RoboDK station: kr30 cnc 042619 3.rdk

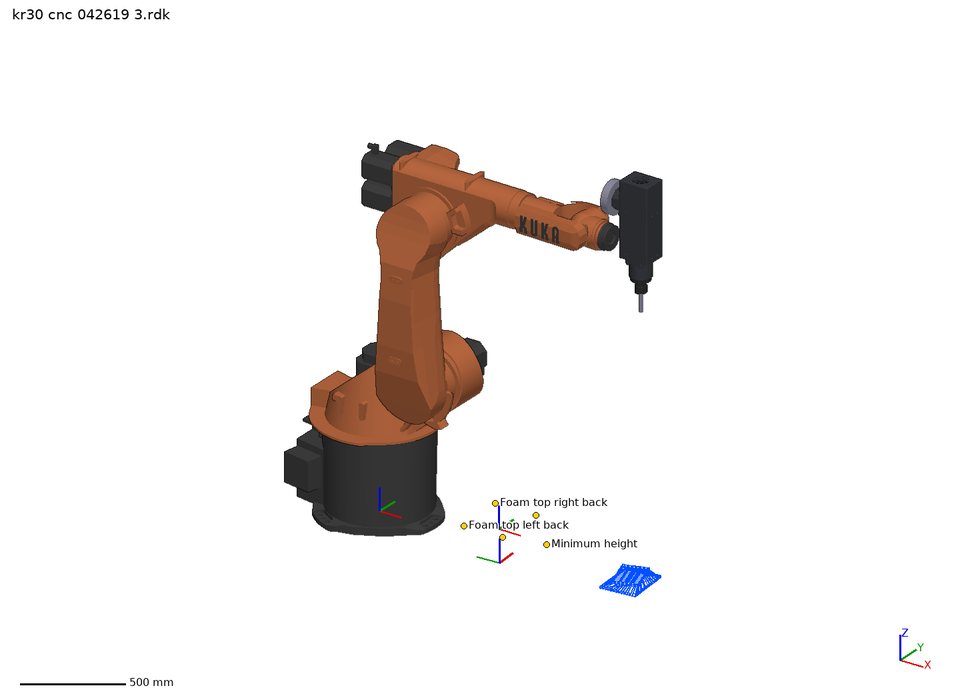
[picture v0: the station drawn from its stored meshes, robots at their saved joint values, targets as dots, program paths as lines]
Station kr30 cnc 042619 3. Poses are relative to the parent item; angles as X-Y-Z fixed-axis rotations.
  - frame KUKA KR 30 HA Base at (0, 0, 0) mm
    - robot KUKA KR 30 HA: 6 axes, payload 30 kg, reach 2033 mm, repeatability 0.05 mm, weight 665 kg
        modified DH rows (alpha deg, a mm, theta deg, d mm): 0, 0, 0, 815; -90, 350, 0, 0; 0, 850, -90, 0; -90, 145, 0, 820; 90, 0, 0, 0; -90, 0, 180, 170
        joint limits [-185, -135, -120, -350, -119, -350] to [185, 35, 158, 350, 119, 350]; home [0, -90, 90, 0, 0, 0]; saved at [0, -90, 90, 0, 0, 0]
      - tool 1/2" End Mill TCP, TCP at (337.71, -2.2, 160.57) mm, size 692.9 x 170 x 256 mm
    - target Foam top left back (Cartesian target) at (1063.86, -826.06, 550.69) mm, rotated rx 159.7 ry 88.57 rz 162.75 deg; joints [48.687, -67.326, 134.977, 54.316, -75.107, -18.491] of KUKA KR 30 HA
    - target Foam top left front (Cartesian target) at (1286.98, -826.06, 550.69) mm, rotated rx 159.7 ry 88.57 rz 162.75 deg; joints [41.175, -60.323, 122.494, 48.236, -69.2, -20.879] of KUKA KR 30 HA
    - target Foam top right front (Cartesian target) at (1280.06, -542.45, 550.69) mm, rotated rx 159.7 ry 88.57 rz 162.75 deg; joints [30.324, -67.933, 136.027, 35.681, -70.54, -13.067] of KUKA KR 30 HA
    - target Foam top right back (Cartesian target) at (1046.63, -542.45, 550.69) mm, rotated rx 159.7 ry 88.57 rz 162.75 deg; joints [37.717, -76.667, 150.322, 42.198, -76.379, -11.394] of KUKA KR 30 HA
    - target Minimum height (Cartesian target) at (1343.09, -542.45, 414.96) mm, rotated rx 159.7 ry 88.57 rz 162.75 deg; joints [28.758, -56.078, 131.986, 32.777, -76.732, -8.072] of KUKA KR 30 HA
  - frame Milling Reference at (1261.16, -812.82, 405.21) mm, rotated rx 0 ry 0 rz 95.1 deg
    - object RhinoCrv at (0, 0, 0) mm
  - frame Frame 3 at (1034.37, -496.81, 391.96) mm
  - program RhinoPart (604 instructions, listed below)
  - machining project RhinoCrv Settings: rotZ(0) | rotX(0)*rotY(0) | rotx(-90)*rotz(270)
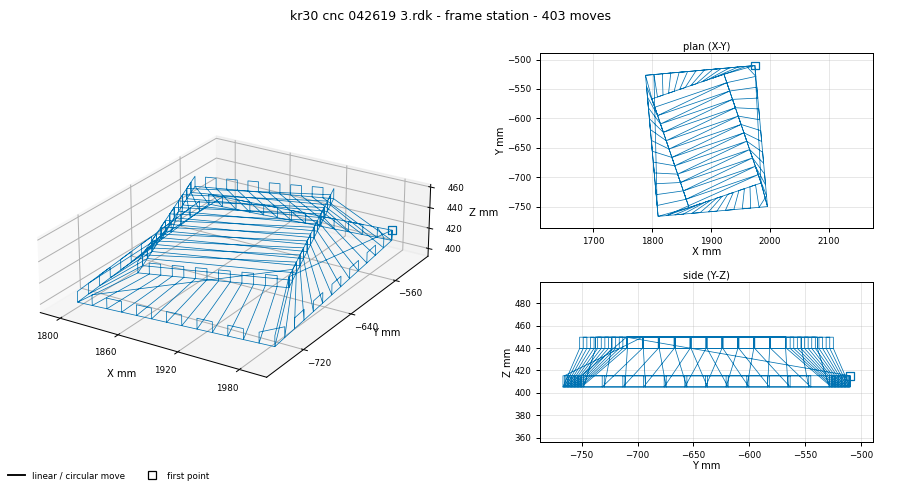
[picture p0: tool path of kr30 cnc 042619 3.rdk in frame station, 403 of 403 moves have a stored position in this frame; points joined in program order, loops and branches not executed]

--- program RhinoPart (robot KUKA KR 30 HA) ---
  Set Ref.: Milling Reference
  Set Tool: 1/2" End Mill TCP
  Show 1/2" End Mill TCP
  Set speed (1000.0 mm/s)
  MoveJ 1 to (238.03, -737.64, 10) mm, rotated rx 0 ry 90 rz 0 deg; joints [38.591, -57.439, 128.954, 40.079, -75.652, -11.779]
  MoveL 2 to (238.03, -737.64, 10) mm, rotated rx 0 ry 90 rz 0 deg; joints [38.591, -57.439, 128.954, 40.079, -75.652, -11.779]
  MoveL 3 to (238.03, -737.64, 0) mm, rotated rx 0 ry 90 rz 0 deg; joints [38.591, -56.76, 128.935, 39.972, -76.157, -11.341]
  MoveL 4 to (238.03, -737.64, 0) mm, rotated rx 0 ry 90 rz 0 deg; joints [38.591, -56.76, 128.935, 39.972, -76.157, -11.341]
  Set speed (50.0 mm/s)
  MoveL 5 to (-2.78, -737.64, 0) mm, rotated rx 0 ry 90 rz 0 deg; joints [46.995, -62.761, 142.501, 47.455, -83.022, -7.54]
  MoveL 6 to (-2.78, -550.89, 0) mm, rotated rx 0 ry 90 rz 0 deg; joints [38.861, -66.566, 151.828, 38.957, -86.312, -2.977]
  MoveL 7 to (238.03, -550.89, 0) mm, rotated rx 0 ry 90 rz 0 deg; joints [30.953, -60.465, 137.205, 31.641, -78.655, -6.911]
  MoveL 8 to (238.03, -737.64, 0) mm, rotated rx 0 ry 90 rz 0 deg; joints [38.591, -56.76, 128.935, 39.972, -76.157, -11.341]
  Set speed (1000.0 mm/s)
  MoveL 9 to (238.03, -737.64, 0) mm, rotated rx 0 ry 90 rz 0 deg; joints [38.591, -56.76, 128.935, 39.972, -76.157, -11.341]
  MoveL 10 to (238.03, -737.64, 10) mm, rotated rx 0 ry 90 rz 0 deg; joints [38.591, -57.439, 128.954, 40.079, -75.652, -11.779]
  Set speed (1000.0 mm/s)
  MoveL 11 to (38.14, -730.32, 44.46) mm, rotated rx 0 ry 90 rz 0 deg; joints [45.091, -65.66, 140.789, 46.066, -79.561, -10.651]
  MoveL 12 to (38.14, -730.32, 34.46) mm, rotated rx 0 ry 90 rz 0 deg; joints [45.091, -64.85, 140.804, 45.96, -80.134, -10.048]
  MoveL 13 to (38.14, -730.32, 34.46) mm, rotated rx 0 ry 90 rz 0 deg; joints [45.091, -64.85, 140.804, 45.96, -80.134, -10.048]
  Set speed (50.0 mm/s)
  MoveL 14 to (7.39, -604.64, 34.46) mm, rotated rx 0 ry 90 rz 0 deg; joints [41.018, -68.705, 148.8, 41.444, -82.543, -6.538]
  MoveL 15 to (197.11, -558.22, 34.46) mm, rotated rx 0 ry 90 rz 0 deg; joints [32.421, -64.255, 139.577, 33.287, -77.649, -7.994]
  MoveL 16 to (227.86, -683.9, 34.46) mm, rotated rx 0 ry 90 rz 0 deg; joints [36.836, -60.65, 132.171, 38.301, -75.305, -11.329]
  MoveL 17 to (38.14, -730.32, 34.46) mm, rotated rx 0 ry 90 rz 0 deg; joints [45.091, -64.85, 140.804, 45.96, -80.134, -10.048]
  Set speed (1000.0 mm/s)
  MoveL 18 to (38.14, -730.32, 34.46) mm, rotated rx 0 ry 90 rz 0 deg; joints [45.091, -64.85, 140.804, 45.96, -80.134, -10.048]
  MoveL 19 to (38.14, -730.32, 44.46) mm, rotated rx 0 ry 90 rz 0 deg; joints [45.091, -65.66, 140.789, 46.066, -79.561, -10.651]
  Set speed (1000.0 mm/s)
  MoveL 20 to (-2.78, -737.64, 10) mm, rotated rx 0 ry 90 rz 0 deg; joints [46.995, -63.616, 142.523, 47.534, -82.46, -8.159]
  MoveL 21 to (-2.78, -737.64, 0) mm, rotated rx 0 ry 90 rz 0 deg; joints [46.995, -62.761, 142.501, 47.455, -83.022, -7.54]
  MoveL 22 to (-2.78, -737.64, 0) mm, rotated rx 0 ry 90 rz 0 deg; joints [46.995, -62.761, 142.501, 47.455, -83.022, -7.54]
  Set speed (50.0 mm/s)
  MoveL 23 to (38.14, -730.32, 34.46) mm, rotated rx 0 ry 90 rz 0 deg; joints [45.091, -64.85, 140.804, 45.96, -80.134, -10.048]
  Set speed (1000.0 mm/s)
  MoveL 24 to (38.14, -730.32, 34.46) mm, rotated rx 0 ry 90 rz 0 deg; joints [45.091, -64.85, 140.804, 45.96, -80.134, -10.048]
  MoveL 25 to (38.14, -730.32, 44.46) mm, rotated rx 0 ry 90 rz 0 deg; joints [45.091, -65.66, 140.789, 46.066, -79.561, -10.651]
  Set speed (1000.0 mm/s)
  MoveL 26 to (227.86, -683.9, 44.46) mm, rotated rx 0 ry 90 rz 0 deg; joints [36.836, -61.347, 132.158, 38.419, -74.748, -11.786]
  MoveL 27 to (227.86, -683.9, 34.46) mm, rotated rx 0 ry 90 rz 0 deg; joints [36.836, -60.65, 132.171, 38.301, -75.305, -11.329]
  MoveL 28 to (227.86, -683.9, 34.46) mm, rotated rx 0 ry 90 rz 0 deg; joints [36.836, -60.65, 132.171, 38.301, -75.305, -11.329]
  Set speed (50.0 mm/s)
  MoveL 29 to (238.03, -737.64, 0) mm, rotated rx 0 ry 90 rz 0 deg; joints [38.591, -56.76, 128.935, 39.972, -76.157, -11.341]
  Set speed (1000.0 mm/s)
  MoveL 30 to (238.03, -737.64, 0) mm, rotated rx 0 ry 90 rz 0 deg; joints [38.591, -56.76, 128.935, 39.972, -76.157, -11.341]
  MoveL 31 to (238.03, -737.64, 10) mm, rotated rx 0 ry 90 rz 0 deg; joints [38.591, -57.439, 128.954, 40.079, -75.652, -11.779]
  Set speed (1000.0 mm/s)
  MoveL 32 to (238.03, -550.89, 10) mm, rotated rx 0 ry 90 rz 0 deg; joints [30.953, -61.24, 137.226, 31.723, -78.013, -7.316]
  MoveL 33 to (238.03, -550.89, 0) mm, rotated rx 0 ry 90 rz 0 deg; joints [30.953, -60.465, 137.205, 31.641, -78.655, -6.911]
  MoveL 34 to (238.03, -550.89, 0) mm, rotated rx 0 ry 90 rz 0 deg; joints [30.953, -60.465, 137.205, 31.641, -78.655, -6.911]
  Set speed (50.0 mm/s)
  MoveL 35 to (197.11, -558.22, 34.46) mm, rotated rx 0 ry 90 rz 0 deg; joints [32.421, -64.255, 139.577, 33.287, -77.649, -7.994]
  Set speed (1000.0 mm/s)
  MoveL 36 to (197.11, -558.22, 34.46) mm, rotated rx 0 ry 90 rz 0 deg; joints [32.421, -64.255, 139.577, 33.287, -77.649, -7.994]
  MoveL 37 to (197.11, -558.22, 44.46) mm, rotated rx 0 ry 90 rz 0 deg; joints [32.421, -65.047, 139.563, 33.387, -76.976, -8.448]
  Set speed (1000.0 mm/s)
  MoveL 38 to (7.39, -604.64, 44.46) mm, rotated rx 0 ry 90 rz 0 deg; joints [41.018, -69.663, 148.783, 41.533, -81.812, -7.19]
  MoveL 39 to (7.39, -604.64, 34.46) mm, rotated rx 0 ry 90 rz 0 deg; joints [41.018, -68.705, 148.8, 41.444, -82.543, -6.538]
  MoveL 40 to (7.39, -604.64, 34.46) mm, rotated rx 0 ry 90 rz 0 deg; joints [41.018, -68.705, 148.8, 41.444, -82.543, -6.538]
  Set speed (50.0 mm/s)
  MoveL 41 to (-2.78, -550.89, 0) mm, rotated rx 0 ry 90 rz 0 deg; joints [38.861, -66.566, 151.828, 38.957, -86.312, -2.977]
  Set speed (1000.0 mm/s)
  MoveL 42 to (-2.78, -550.89, 0) mm, rotated rx 0 ry 90 rz 0 deg; joints [38.861, -66.566, 151.828, 38.957, -86.312, -2.977]
  MoveL 43 to (-2.78, -550.89, 10) mm, rotated rx 0 ry 90 rz 0 deg; joints [38.861, -67.618, 151.855, 39.003, -85.515, -3.624]
  Set speed (1000.0 mm/s)
  MoveL 44 to (219.51, -550.89, 10) mm, rotated rx 0 ry 90 rz 0 deg; joints [31.458, -61.784, 138.427, 32.162, -78.635, -7.064]
  MoveL 45 to (219.51, -550.89, 0) mm, rotated rx 0 ry 90 rz 0 deg; joints [31.458, -60.992, 138.406, 32.082, -79.288, -6.646]
  MoveL 46 to (219.51, -550.89, 0) mm, rotated rx 0 ry 90 rz 0 deg; joints [31.458, -60.992, 138.406, 32.082, -79.288, -6.646]
  Set speed (50.0 mm/s)
  MoveL 47 to (182.51, -561.79, 34.46) mm, rotated rx 0 ry 90 rz 0 deg; joints [33.008, -64.633, 140.355, 33.835, -78.065, -7.893]
  Set speed (1000.0 mm/s)
  MoveL 48 to (182.51, -561.79, 34.46) mm, rotated rx 0 ry 90 rz 0 deg; joints [33.008, -64.633, 140.355, 33.835, -78.065, -7.893]
  MoveL 49 to (182.51, -561.79, 44.46) mm, rotated rx 0 ry 90 rz 0 deg; joints [33.008, -65.436, 140.34, 33.934, -77.385, -8.359]
  Set speed (1000.0 mm/s)
  MoveL 50 to (167.92, -565.36, 44.46) mm, rotated rx 0 ry 90 rz 0 deg; joints [33.607, -65.82, 141.107, 34.494, -77.789, -8.269]
  MoveL 51 to (167.92, -565.36, 34.46) mm, rotated rx 0 ry 90 rz 0 deg; joints [33.607, -65.005, 141.123, 34.395, -78.474, -7.789]
  MoveL 52 to (167.92, -565.36, 34.46) mm, rotated rx 0 ry 90 rz 0 deg; joints [33.607, -65.005, 141.123, 34.395, -78.474, -7.789]
  Set speed (50.0 mm/s)
  MoveL 53 to (200.98, -550.89, 0) mm, rotated rx 0 ry 90 rz 0 deg; joints [31.977, -61.51, 139.595, 32.54, -79.913, -6.376]
  Set speed (1000.0 mm/s)
  MoveL 54 to (200.98, -550.89, 0) mm, rotated rx 0 ry 90 rz 0 deg; joints [31.977, -61.51, 139.595, 32.54, -79.913, -6.376]
  MoveL 55 to (200.98, -550.89, 10) mm, rotated rx 0 ry 90 rz 0 deg; joints [31.977, -62.319, 139.616, 32.618, -79.25, -6.807]
  Set speed (1000.0 mm/s)
  MoveL 56 to (182.46, -550.89, 10) mm, rotated rx 0 ry 90 rz 0 deg; joints [32.512, -62.846, 140.793, 33.094, -79.858, -6.547]
  MoveL 57 to (182.46, -550.89, 0) mm, rotated rx 0 ry 90 rz 0 deg; joints [32.512, -62.019, 140.771, 33.018, -80.532, -6.101]
  MoveL 58 to (182.46, -550.89, 0) mm, rotated rx 0 ry 90 rz 0 deg; joints [32.512, -62.019, 140.771, 33.018, -80.532, -6.101]
  Set speed (50.0 mm/s)
  MoveL 59 to (153.32, -568.93, 34.46) mm, rotated rx 0 ry 90 rz 0 deg; joints [34.218, -65.371, 141.879, 34.968, -78.876, -7.684]
  Set speed (1000.0 mm/s)
  MoveL 60 to (153.32, -568.93, 34.46) mm, rotated rx 0 ry 90 rz 0 deg; joints [34.218, -65.371, 141.879, 34.968, -78.876, -7.684]
  MoveL 61 to (153.32, -568.93, 44.46) mm, rotated rx 0 ry 90 rz 0 deg; joints [34.218, -66.198, 141.863, 35.066, -78.187, -8.177]
  Set speed (1000.0 mm/s)
  MoveL 62 to (138.73, -572.5, 44.46) mm, rotated rx 0 ry 90 rz 0 deg; joints [34.841, -66.57, 142.608, 35.651, -78.578, -8.084]
  MoveL 63 to (138.73, -572.5, 34.46) mm, rotated rx 0 ry 90 rz 0 deg; joints [34.841, -65.731, 142.623, 35.554, -79.273, -7.577]
  MoveL 64 to (138.73, -572.5, 34.46) mm, rotated rx 0 ry 90 rz 0 deg; joints [34.841, -65.731, 142.623, 35.554, -79.273, -7.577]
  Set speed (50.0 mm/s)
  MoveL 65 to (163.93, -550.89, 0) mm, rotated rx 0 ry 90 rz 0 deg; joints [33.063, -62.519, 141.935, 33.514, -81.145, -5.821]
  Set speed (1000.0 mm/s)
  MoveL 66 to (163.93, -550.89, 0) mm, rotated rx 0 ry 90 rz 0 deg; joints [33.063, -62.519, 141.935, 33.514, -81.145, -5.821]
  MoveL 67 to (163.93, -550.89, 10) mm, rotated rx 0 ry 90 rz 0 deg; joints [33.063, -63.364, 141.957, 33.588, -80.459, -6.282]
  Set speed (1000.0 mm/s)
  MoveL 68 to (145.41, -550.89, 10) mm, rotated rx 0 ry 90 rz 0 deg; joints [33.631, -63.874, 143.108, 34.101, -81.052, -6.012]
  MoveL 69 to (145.41, -550.89, 0) mm, rotated rx 0 ry 90 rz 0 deg; joints [33.631, -63.009, 143.086, 34.03, -81.75, -5.534]
  MoveL 70 to (145.41, -550.89, 0) mm, rotated rx 0 ry 90 rz 0 deg; joints [33.631, -63.009, 143.086, 34.03, -81.75, -5.534]
  Set speed (50.0 mm/s)
  MoveL 71 to (124.14, -576.07, 34.46) mm, rotated rx 0 ry 90 rz 0 deg; joints [35.476, -66.086, 143.357, 36.153, -79.663, -7.469]
  Set speed (1000.0 mm/s)
  MoveL 72 to (124.14, -576.07, 34.46) mm, rotated rx 0 ry 90 rz 0 deg; joints [35.476, -66.086, 143.357, 36.153, -79.663, -7.469]
  MoveL 73 to (124.14, -576.07, 44.46) mm, rotated rx 0 ry 90 rz 0 deg; joints [35.476, -66.937, 143.341, 36.249, -78.964, -7.99]
  Set speed (1000.0 mm/s)
  MoveL 74 to (109.54, -579.64, 44.46) mm, rotated rx 0 ry 90 rz 0 deg; joints [36.124, -67.299, 144.063, 36.861, -79.343, -7.894]
  MoveL 75 to (109.54, -579.64, 34.46) mm, rotated rx 0 ry 90 rz 0 deg; joints [36.124, -66.434, 144.079, 36.765, -80.047, -7.358]
  MoveL 76 to (109.54, -579.64, 34.46) mm, rotated rx 0 ry 90 rz 0 deg; joints [36.124, -66.434, 144.079, 36.765, -80.047, -7.358]
  Set speed (50.0 mm/s)
  MoveL 77 to (126.89, -550.89, 0) mm, rotated rx 0 ry 90 rz 0 deg; joints [34.216, -63.49, 144.224, 34.567, -82.349, -5.241]
  Set speed (1000.0 mm/s)
  MoveL 78 to (126.89, -550.89, 0) mm, rotated rx 0 ry 90 rz 0 deg; joints [34.216, -63.49, 144.224, 34.567, -82.349, -5.241]
  MoveL 79 to (126.89, -550.89, 10) mm, rotated rx 0 ry 90 rz 0 deg; joints [34.216, -64.375, 144.247, 34.635, -81.639, -5.736]
  Set speed (1000.0 mm/s)
  MoveL 80 to (108.36, -550.89, 10) mm, rotated rx 0 ry 90 rz 0 deg; joints [34.819, -64.867, 145.373, 35.19, -82.218, -5.455]
  MoveL 81 to (108.36, -550.89, 0) mm, rotated rx 0 ry 90 rz 0 deg; joints [34.819, -63.961, 145.35, 35.124, -82.939, -4.942]
  MoveL 82 to (108.36, -550.89, 0) mm, rotated rx 0 ry 90 rz 0 deg; joints [34.819, -63.961, 145.35, 35.124, -82.939, -4.942]
  Set speed (50.0 mm/s)
  MoveL 83 to (94.95, -583.21, 34.46) mm, rotated rx 0 ry 90 rz 0 deg; joints [36.784, -66.777, 144.79, 37.391, -80.425, -7.246]
  Set speed (1000.0 mm/s)
  MoveL 84 to (94.95, -583.21, 34.46) mm, rotated rx 0 ry 90 rz 0 deg; joints [36.784, -66.777, 144.79, 37.391, -80.425, -7.246]
  MoveL 85 to (94.95, -583.21, 44.46) mm, rotated rx 0 ry 90 rz 0 deg; joints [36.784, -67.654, 144.774, 37.486, -79.715, -7.797]
  Set speed (1000.0 mm/s)
  MoveL 86 to (80.36, -586.78, 44.46) mm, rotated rx 0 ry 90 rz 0 deg; joints [37.456, -68.004, 145.472, 38.125, -80.082, -7.699]
  MoveL 87 to (80.36, -586.78, 34.46) mm, rotated rx 0 ry 90 rz 0 deg; joints [37.456, -67.114, 145.489, 38.031, -80.795, -7.132]
  MoveL 88 to (80.36, -586.78, 34.46) mm, rotated rx 0 ry 90 rz 0 deg; joints [37.456, -67.114, 145.489, 38.031, -80.795, -7.132]
  Set speed (50.0 mm/s)
  MoveL 89 to (89.84, -550.89, 0) mm, rotated rx 0 ry 90 rz 0 deg; joints [35.441, -64.422, 146.462, 35.704, -83.523, -4.635]
  Set speed (1000.0 mm/s)
  MoveL 90 to (89.84, -550.89, 0) mm, rotated rx 0 ry 90 rz 0 deg; joints [35.441, -64.422, 146.462, 35.704, -83.523, -4.635]
  MoveL 91 to (89.84, -550.89, 10) mm, rotated rx 0 ry 90 rz 0 deg; joints [35.441, -65.35, 146.486, 35.767, -82.789, -5.167]
  Set speed (1000.0 mm/s)
  MoveL 92 to (71.31, -550.89, 10) mm, rotated rx 0 ry 90 rz 0 deg; joints [36.083, -65.823, 147.587, 36.366, -83.352, -4.873]
  MoveL 93 to (71.31, -550.89, 0) mm, rotated rx 0 ry 90 rz 0 deg; joints [36.083, -64.872, 147.562, 36.306, -84.098, -4.321]
  MoveL 94 to (71.31, -550.89, 0) mm, rotated rx 0 ry 90 rz 0 deg; joints [36.083, -64.872, 147.562, 36.306, -84.098, -4.321]
  Set speed (50.0 mm/s)
  MoveL 95 to (65.76, -590.35, 34.46) mm, rotated rx 0 ry 90 rz 0 deg; joints [38.142, -67.445, 146.176, 38.685, -81.159, -7.016]
  Set speed (1000.0 mm/s)
  MoveL 96 to (65.76, -590.35, 34.46) mm, rotated rx 0 ry 90 rz 0 deg; joints [38.142, -67.445, 146.176, 38.685, -81.159, -7.016]
  MoveL 97 to (65.76, -590.35, 44.46) mm, rotated rx 0 ry 90 rz 0 deg; joints [38.142, -68.348, 146.159, 38.778, -80.441, -7.599]
  Set speed (1000.0 mm/s)
  MoveL 98 to (51.17, -593.92, 44.46) mm, rotated rx 0 ry 90 rz 0 deg; joints [38.841, -68.686, 146.834, 39.445, -80.794, -7.498]
  MoveL 99 to (51.17, -593.92, 34.46) mm, rotated rx 0 ry 90 rz 0 deg; joints [38.841, -67.769, 146.85, 39.353, -81.516, -6.899]
  MoveL 100 to (51.17, -593.92, 34.46) mm, rotated rx 0 ry 90 rz 0 deg; joints [38.841, -67.769, 146.85, 39.353, -81.516, -6.899]
  Set speed (50.0 mm/s)
  MoveL 101 to (52.79, -550.89, 0) mm, rotated rx 0 ry 90 rz 0 deg; joints [36.745, -65.312, 148.649, 36.931, -84.665, -3.998]
  Set speed (1000.0 mm/s)
  MoveL 102 to (52.79, -550.89, 0) mm, rotated rx 0 ry 90 rz 0 deg; joints [36.745, -65.312, 148.649, 36.931, -84.665, -3.998]
  MoveL 103 to (52.79, -550.89, 10) mm, rotated rx 0 ry 90 rz 0 deg; joints [36.745, -66.287, 148.674, 36.988, -83.906, -4.572]
  Set speed (1000.0 mm/s)
  MoveL 104 to (34.27, -550.89, 10) mm, rotated rx 0 ry 90 rz 0 deg; joints [37.428, -66.741, 149.748, 37.635, -84.452, -4.264]
  MoveL 105 to (34.27, -550.89, 0) mm, rotated rx 0 ry 90 rz 0 deg; joints [37.428, -65.742, 149.722, 37.581, -85.223, -3.667]
  MoveL 106 to (34.27, -550.89, 0) mm, rotated rx 0 ry 90 rz 0 deg; joints [37.428, -65.742, 149.722, 37.581, -85.223, -3.667]
  Set speed (50.0 mm/s)
  MoveL 107 to (36.58, -597.5, 34.46) mm, rotated rx 0 ry 90 rz 0 deg; joints [39.553, -68.088, 147.513, 40.036, -81.865, -6.78]
  Set speed (1000.0 mm/s)
  MoveL 108 to (36.58, -597.5, 34.46) mm, rotated rx 0 ry 90 rz 0 deg; joints [39.553, -68.088, 147.513, 40.036, -81.865, -6.78]
  MoveL 109 to (36.58, -597.5, 44.46) mm, rotated rx 0 ry 90 rz 0 deg; joints [39.553, -69.018, 147.496, 40.127, -81.14, -7.397]
  Set speed (1000.0 mm/s)
  MoveL 110 to (21.98, -601.07, 44.46) mm, rotated rx 0 ry 90 rz 0 deg; joints [40.279, -69.344, 148.146, 40.823, -81.48, -7.294]
  MoveL 111 to (21.98, -601.07, 34.46) mm, rotated rx 0 ry 90 rz 0 deg; joints [40.279, -68.4, 148.163, 40.733, -82.208, -6.659]
  MoveL 112 to (21.98, -601.07, 34.46) mm, rotated rx 0 ry 90 rz 0 deg; joints [40.279, -68.4, 148.163, 40.733, -82.208, -6.659]
  Set speed (50.0 mm/s)
  MoveL 113 to (15.74, -550.89, 0) mm, rotated rx 0 ry 90 rz 0 deg; joints [38.133, -66.16, 150.782, 38.256, -85.772, -3.327]
  Set speed (1000.0 mm/s)
  MoveL 114 to (15.74, -550.89, 0) mm, rotated rx 0 ry 90 rz 0 deg; joints [38.133, -66.16, 150.782, 38.256, -85.772, -3.327]
  MoveL 115 to (15.74, -550.89, 10) mm, rotated rx 0 ry 90 rz 0 deg; joints [38.133, -67.185, 150.808, 38.306, -84.988, -3.948]
  Set speed (1000.0 mm/s)
  MoveL 116 to (238.03, -565.26, 10) mm, rotated rx 0 ry 90 rz 0 deg; joints [31.592, -60.983, 136.658, 32.405, -77.834, -7.619]
  MoveL 117 to (238.03, -565.26, 0) mm, rotated rx 0 ry 90 rz 0 deg; joints [31.592, -60.215, 136.637, 32.321, -78.464, -7.211]
  MoveL 118 to (238.03, -565.26, 0) mm, rotated rx 0 ry 90 rz 0 deg; joints [31.592, -60.215, 136.637, 32.321, -78.464, -7.211]
  Set speed (50.0 mm/s)
  MoveL 119 to (199.47, -567.88, 34.46) mm, rotated rx 0 ry 90 rz 0 deg; joints [32.788, -63.992, 139.035, 33.694, -77.468, -8.232]
  Set speed (1000.0 mm/s)
  MoveL 120 to (199.47, -567.88, 34.46) mm, rotated rx 0 ry 90 rz 0 deg; joints [32.788, -63.992, 139.035, 33.694, -77.468, -8.232]
  MoveL 121 to (199.47, -567.88, 44.46) mm, rotated rx 0 ry 90 rz 0 deg; joints [32.788, -64.776, 139.02, 33.795, -76.805, -8.687]
  Set speed (1000.0 mm/s)
  MoveL 122 to (201.84, -577.55, 44.46) mm, rotated rx 0 ry 90 rz 0 deg; joints [33.151, -64.502, 138.472, 34.199, -76.633, -8.929]
  MoveL 123 to (201.84, -577.55, 34.46) mm, rotated rx 0 ry 90 rz 0 deg; joints [33.151, -63.726, 138.487, 34.097, -77.287, -8.473]
  MoveL 124 to (201.84, -577.55, 34.46) mm, rotated rx 0 ry 90 rz 0 deg; joints [33.151, -63.726, 138.487, 34.097, -77.287, -8.473]
  Set speed (50.0 mm/s)
  MoveL 125 to (238.03, -579.62, 0) mm, rotated rx 0 ry 90 rz 0 deg; joints [32.222, -59.959, 136.058, 32.995, -78.273, -7.518]
  Set speed (1000.0 mm/s)
  MoveL 126 to (238.03, -579.62, 0) mm, rotated rx 0 ry 90 rz 0 deg; joints [32.222, -59.959, 136.058, 32.995, -78.273, -7.518]
  MoveL 127 to (238.03, -579.62, 10) mm, rotated rx 0 ry 90 rz 0 deg; joints [32.222, -60.719, 136.078, 33.081, -77.653, -7.93]
  Set speed (1000.0 mm/s)
  MoveL 128 to (238.03, -593.99, 10) mm, rotated rx 0 ry 90 rz 0 deg; joints [32.843, -60.45, 135.487, 33.75, -77.472, -8.247]
  MoveL 129 to (238.03, -593.99, 0) mm, rotated rx 0 ry 90 rz 0 deg; joints [32.843, -59.697, 135.467, 33.662, -78.081, -7.831]
  MoveL 130 to (238.03, -593.99, 0) mm, rotated rx 0 ry 90 rz 0 deg; joints [32.843, -59.697, 135.467, 33.662, -78.081, -7.831]
  Set speed (50.0 mm/s)
  MoveL 131 to (204.2, -587.22, 34.46) mm, rotated rx 0 ry 90 rz 0 deg; joints [33.509, -63.458, 137.935, 34.496, -77.106, -8.718]
  Set speed (1000.0 mm/s)
  MoveL 132 to (204.2, -587.22, 34.46) mm, rotated rx 0 ry 90 rz 0 deg; joints [33.509, -63.458, 137.935, 34.496, -77.106, -8.718]
  MoveL 133 to (204.2, -587.22, 44.46) mm, rotated rx 0 ry 90 rz 0 deg; joints [33.509, -64.226, 137.921, 34.6, -76.462, -9.174]
  Set speed (1000.0 mm/s)
  MoveL 134 to (206.57, -596.89, 44.46) mm, rotated rx 0 ry 90 rz 0 deg; joints [33.862, -63.948, 137.364, 34.997, -76.29, -9.421]
  MoveL 135 to (206.57, -596.89, 34.46) mm, rotated rx 0 ry 90 rz 0 deg; joints [33.862, -63.187, 137.379, 34.891, -76.926, -8.965]
  MoveL 136 to (206.57, -596.89, 34.46) mm, rotated rx 0 ry 90 rz 0 deg; joints [33.862, -63.187, 137.379, 34.891, -76.926, -8.965]
  Set speed (50.0 mm/s)
  MoveL 137 to (238.03, -608.35, 0) mm, rotated rx 0 ry 90 rz 0 deg; joints [33.455, -59.43, 134.864, 34.322, -77.888, -8.152]
  Set speed (1000.0 mm/s)
  MoveL 138 to (238.03, -608.35, 0) mm, rotated rx 0 ry 90 rz 0 deg; joints [33.455, -59.43, 134.864, 34.322, -77.888, -8.152]
  MoveL 139 to (238.03, -608.35, 10) mm, rotated rx 0 ry 90 rz 0 deg; joints [33.455, -60.174, 134.884, 34.412, -77.29, -8.571]
  Set speed (1000.0 mm/s)
  MoveL 140 to (238.03, -622.72, 10) mm, rotated rx 0 ry 90 rz 0 deg; joints [34.059, -59.893, 134.27, 35.067, -77.108, -8.901]
  MoveL 141 to (238.03, -622.72, 0) mm, rotated rx 0 ry 90 rz 0 deg; joints [34.059, -59.156, 134.25, 34.975, -77.696, -8.479]
  MoveL 142 to (238.03, -622.72, 0) mm, rotated rx 0 ry 90 rz 0 deg; joints [34.059, -59.156, 134.25, 34.975, -77.696, -8.479]
  Set speed (50.0 mm/s)
  MoveL 143 to (208.93, -606.55, 34.46) mm, rotated rx 0 ry 90 rz 0 deg; joints [34.21, -62.915, 136.818, 35.283, -76.745, -9.216]
  Set speed (1000.0 mm/s)
  MoveL 144 to (208.93, -606.55, 34.46) mm, rotated rx 0 ry 90 rz 0 deg; joints [34.21, -62.915, 136.818, 35.283, -76.745, -9.216]
  MoveL 145 to (208.93, -606.55, 44.46) mm, rotated rx 0 ry 90 rz 0 deg; joints [34.21, -63.668, 136.804, 35.39, -76.119, -9.672]
  Set speed (1000.0 mm/s)
  MoveL 146 to (211.3, -616.22, 44.46) mm, rotated rx 0 ry 90 rz 0 deg; joints [34.554, -63.385, 136.238, 35.78, -75.947, -9.926]
  MoveL 147 to (211.3, -616.22, 34.46) mm, rotated rx 0 ry 90 rz 0 deg; joints [34.554, -62.639, 136.252, 35.672, -76.564, -9.469]
  MoveL 148 to (211.3, -616.22, 34.46) mm, rotated rx 0 ry 90 rz 0 deg; joints [34.554, -62.639, 136.252, 35.672, -76.564, -9.469]
  Set speed (50.0 mm/s)
  MoveL 149 to (238.03, -637.08, 0) mm, rotated rx 0 ry 90 rz 0 deg; joints [34.655, -58.877, 133.625, 35.622, -77.503, -8.813]
  Set speed (1000.0 mm/s)
  MoveL 150 to (238.03, -637.08, 0) mm, rotated rx 0 ry 90 rz 0 deg; joints [34.655, -58.877, 133.625, 35.622, -77.503, -8.813]
  MoveL 151 to (238.03, -637.08, 10) mm, rotated rx 0 ry 90 rz 0 deg; joints [34.655, -59.606, 133.645, 35.716, -76.926, -9.238]
  Set speed (1000.0 mm/s)
  MoveL 152 to (238.03, -651.45, 10) mm, rotated rx 0 ry 90 rz 0 deg; joints [35.242, -59.314, 133.008, 36.358, -76.744, -9.581]
  MoveL 153 to (238.03, -651.45, 0) mm, rotated rx 0 ry 90 rz 0 deg; joints [35.242, -58.592, 132.988, 36.262, -77.31, -9.154]
  MoveL 154 to (238.03, -651.45, 0) mm, rotated rx 0 ry 90 rz 0 deg; joints [35.242, -58.592, 132.988, 36.262, -77.31, -9.154]
  Set speed (50.0 mm/s)
  MoveL 155 to (213.66, -625.89, 34.46) mm, rotated rx 0 ry 90 rz 0 deg; joints [34.893, -62.362, 135.683, 36.057, -76.384, -9.726]
  Set speed (1000.0 mm/s)
  MoveL 156 to (213.66, -625.89, 34.46) mm, rotated rx 0 ry 90 rz 0 deg; joints [34.893, -62.362, 135.683, 36.057, -76.384, -9.726]
  MoveL 157 to (213.66, -625.89, 44.46) mm, rotated rx 0 ry 90 rz 0 deg; joints [34.893, -63.101, 135.669, 36.167, -75.776, -10.183]
  Set speed (1000.0 mm/s)
  MoveL 158 to (216.03, -635.56, 44.46) mm, rotated rx 0 ry 90 rz 0 deg; joints [35.228, -62.814, 135.095, 36.55, -75.604, -10.443]
  MoveL 159 to (216.03, -635.56, 34.46) mm, rotated rx 0 ry 90 rz 0 deg; joints [35.228, -62.082, 135.109, 36.439, -76.204, -9.985]
  MoveL 160 to (216.03, -635.56, 34.46) mm, rotated rx 0 ry 90 rz 0 deg; joints [35.228, -62.082, 135.109, 36.439, -76.204, -9.985]
  Set speed (50.0 mm/s)
  MoveL 161 to (238.03, -665.81, 0) mm, rotated rx 0 ry 90 rz 0 deg; joints [35.821, -58.301, 132.34, 36.896, -77.117, -9.502]
  Set speed (1000.0 mm/s)
  MoveL 162 to (238.03, -665.81, 0) mm, rotated rx 0 ry 90 rz 0 deg; joints [35.821, -58.301, 132.34, 36.896, -77.117, -9.502]
  MoveL 163 to (238.03, -665.81, 10) mm, rotated rx 0 ry 90 rz 0 deg; joints [35.821, -59.015, 132.36, 36.994, -76.561, -9.931]
  Set speed (1000.0 mm/s)
  MoveL 164 to (238.03, -680.18, 10) mm, rotated rx 0 ry 90 rz 0 deg; joints [36.391, -58.711, 131.701, 37.623, -76.379, -10.288]
  MoveL 165 to (238.03, -680.18, 0) mm, rotated rx 0 ry 90 rz 0 deg; joints [36.391, -58.004, 131.681, 37.524, -76.924, -9.856]
  MoveL 166 to (238.03, -680.18, 0) mm, rotated rx 0 ry 90 rz 0 deg; joints [36.391, -58.004, 131.681, 37.524, -76.924, -9.856]
  Set speed (50.0 mm/s)
  MoveL 167 to (218.4, -645.22, 34.46) mm, rotated rx 0 ry 90 rz 0 deg; joints [35.558, -61.8, 134.53, 36.817, -76.024, -10.248]
  Set speed (1000.0 mm/s)
  MoveL 168 to (218.4, -645.22, 34.46) mm, rotated rx 0 ry 90 rz 0 deg; joints [35.558, -61.8, 134.53, 36.817, -76.024, -10.248]
  MoveL 169 to (218.4, -645.22, 44.46) mm, rotated rx 0 ry 90 rz 0 deg; joints [35.558, -62.525, 134.516, 36.93, -75.433, -10.705]
  Set speed (1000.0 mm/s)
  MoveL 170 to (220.76, -654.89, 44.46) mm, rotated rx 0 ry 90 rz 0 deg; joints [35.884, -62.234, 133.933, 37.307, -75.262, -10.971]
  MoveL 171 to (220.76, -654.89, 34.46) mm, rotated rx 0 ry 90 rz 0 deg; joints [35.884, -61.516, 133.947, 37.193, -75.844, -10.514]
  MoveL 172 to (220.76, -654.89, 34.46) mm, rotated rx 0 ry 90 rz 0 deg; joints [35.884, -61.516, 133.947, 37.193, -75.844, -10.514]
  Set speed (50.0 mm/s)
  MoveL 173 to (238.03, -694.54, 0) mm, rotated rx 0 ry 90 rz 0 deg; joints [36.953, -57.701, 131.011, 38.145, -76.732, -10.218]
  Set speed (1000.0 mm/s)
  MoveL 174 to (238.03, -694.54, 0) mm, rotated rx 0 ry 90 rz 0 deg; joints [36.953, -57.701, 131.011, 38.145, -76.732, -10.218]
  MoveL 175 to (238.03, -694.54, 10) mm, rotated rx 0 ry 90 rz 0 deg; joints [36.953, -58.402, 131.03, 38.246, -76.197, -10.651]
  Set speed (1000.0 mm/s)
  MoveL 176 to (238.03, -708.91, 10) mm, rotated rx 0 ry 90 rz 0 deg; joints [37.507, -58.086, 130.349, 38.863, -76.015, -11.02]
  MoveL 177 to (238.03, -708.91, 0) mm, rotated rx 0 ry 90 rz 0 deg; joints [37.507, -57.393, 130.33, 38.76, -76.54, -10.586]
  MoveL 178 to (238.03, -708.91, 0) mm, rotated rx 0 ry 90 rz 0 deg; joints [37.507, -57.393, 130.33, 38.76, -76.54, -10.586]
  Set speed (50.0 mm/s)
  MoveL 179 to (223.13, -664.56, 34.46) mm, rotated rx 0 ry 90 rz 0 deg; joints [36.205, -61.23, 133.359, 37.565, -75.664, -10.783]
  Set speed (1000.0 mm/s)
  MoveL 180 to (223.13, -664.56, 34.46) mm, rotated rx 0 ry 90 rz 0 deg; joints [36.205, -61.23, 133.359, 37.565, -75.664, -10.783]
  MoveL 181 to (223.13, -664.56, 44.46) mm, rotated rx 0 ry 90 rz 0 deg; joints [36.205, -61.94, 133.346, 37.68, -75.09, -11.24]
  Set speed (1000.0 mm/s)
  MoveL 182 to (225.49, -674.23, 44.46) mm, rotated rx 0 ry 90 rz 0 deg; joints [36.522, -61.645, 132.754, 38.051, -74.919, -11.511]
  MoveL 183 to (225.49, -674.23, 34.46) mm, rotated rx 0 ry 90 rz 0 deg; joints [36.522, -60.941, 132.768, 37.935, -75.484, -11.054]
  MoveL 184 to (225.49, -674.23, 34.46) mm, rotated rx 0 ry 90 rz 0 deg; joints [36.522, -60.941, 132.768, 37.935, -75.484, -11.054]
  Set speed (50.0 mm/s)
  MoveL 185 to (238.03, -723.28, 0) mm, rotated rx 0 ry 90 rz 0 deg; joints [38.053, -57.08, 129.638, 39.369, -76.348, -10.96]
  Set speed (1000.0 mm/s)
  MoveL 186 to (238.03, -723.28, 0) mm, rotated rx 0 ry 90 rz 0 deg; joints [38.053, -57.08, 129.638, 39.369, -76.348, -10.96]
  MoveL 187 to (238.03, -723.28, 10) mm, rotated rx 0 ry 90 rz 0 deg; joints [38.053, -57.765, 129.657, 39.474, -75.833, -11.396]
  Set speed (1000.0 mm/s)
  MoveL 188 to (219.51, -737.64, 10) mm, rotated rx 0 ry 90 rz 0 deg; joints [39.147, -57.967, 130.091, 40.542, -76.229, -11.509]
  MoveL 189 to (219.51, -737.64, 0) mm, rotated rx 0 ry 90 rz 0 deg; joints [39.147, -57.276, 130.072, 40.437, -76.739, -11.061]
  MoveL 190 to (219.51, -737.64, 0) mm, rotated rx 0 ry 90 rz 0 deg; joints [39.147, -57.276, 130.072, 40.437, -76.739, -11.061]
  Set speed (50.0 mm/s)
  MoveL 191 to (213.26, -687.47, 34.46) mm, rotated rx 0 ry 90 rz 0 deg; joints [37.412, -61.009, 132.908, 38.824, -75.713, -11.232]
  Set speed (1000.0 mm/s)
  MoveL 192 to (213.26, -687.47, 34.46) mm, rotated rx 0 ry 90 rz 0 deg; joints [37.412, -61.009, 132.908, 38.824, -75.713, -11.232]
  MoveL 193 to (213.26, -687.47, 44.46) mm, rotated rx 0 ry 90 rz 0 deg; joints [37.412, -61.715, 132.894, 38.941, -75.153, -11.699]
  Set speed (1000.0 mm/s)
  MoveL 194 to (198.67, -691.04, 44.46) mm, rotated rx 0 ry 90 rz 0 deg; joints [37.997, -62.077, 133.619, 39.474, -75.552, -11.611]
  MoveL 195 to (198.67, -691.04, 34.46) mm, rotated rx 0 ry 90 rz 0 deg; joints [37.997, -61.363, 133.633, 39.357, -76.114, -11.135]
  MoveL 196 to (198.67, -691.04, 34.46) mm, rotated rx 0 ry 90 rz 0 deg; joints [37.997, -61.363, 133.633, 39.357, -76.114, -11.135]
  Set speed (50.0 mm/s)
  MoveL 197 to (200.98, -737.64, 0) mm, rotated rx 0 ry 90 rz 0 deg; joints [39.717, -57.784, 131.194, 40.919, -77.313, -10.779]
  Set speed (1000.0 mm/s)
  MoveL 198 to (200.98, -737.64, 0) mm, rotated rx 0 ry 90 rz 0 deg; joints [39.717, -57.784, 131.194, 40.919, -77.313, -10.779]
  MoveL 199 to (200.98, -737.64, 10) mm, rotated rx 0 ry 90 rz 0 deg; joints [39.717, -58.486, 131.213, 41.022, -76.797, -11.238]
  Set speed (1000.0 mm/s)
  MoveL 200 to (182.46, -737.64, 10) mm, rotated rx 0 ry 90 rz 0 deg; joints [40.301, -58.997, 132.319, 41.519, -77.357, -10.966]
  MoveL 201 to (182.46, -737.64, 0) mm, rotated rx 0 ry 90 rz 0 deg; joints [40.301, -58.282, 132.3, 41.418, -77.878, -10.495]
  MoveL 202 to (182.46, -737.64, 0) mm, rotated rx 0 ry 90 rz 0 deg; joints [40.301, -58.282, 132.3, 41.418, -77.878, -10.495]
  Set speed (50.0 mm/s)
  MoveL 203 to (184.08, -694.61, 34.46) mm, rotated rx 0 ry 90 rz 0 deg; joints [38.592, -61.711, 134.346, 39.902, -76.51, -11.037]
  Set speed (1000.0 mm/s)
  MoveL 204 to (184.08, -694.61, 34.46) mm, rotated rx 0 ry 90 rz 0 deg; joints [38.592, -61.711, 134.346, 39.902, -76.51, -11.037]
  MoveL 205 to (184.08, -694.61, 44.46) mm, rotated rx 0 ry 90 rz 0 deg; joints [38.592, -62.433, 134.332, 40.017, -75.946, -11.524]
  Set speed (1000.0 mm/s)
  MoveL 206 to (169.48, -698.18, 44.46) mm, rotated rx 0 ry 90 rz 0 deg; joints [39.197, -62.783, 135.033, 40.572, -76.334, -11.437]
  MoveL 207 to (169.48, -698.18, 34.46) mm, rotated rx 0 ry 90 rz 0 deg; joints [39.197, -62.052, 135.047, 40.457, -76.9, -10.939]
  MoveL 208 to (169.48, -698.18, 34.46) mm, rotated rx 0 ry 90 rz 0 deg; joints [39.197, -62.052, 135.047, 40.457, -76.9, -10.939]
  Set speed (50.0 mm/s)
  MoveL 209 to (163.93, -737.64, 0) mm, rotated rx 0 ry 90 rz 0 deg; joints [40.899, -58.772, 133.39, 41.935, -78.434, -10.21]
  Set speed (1000.0 mm/s)
  MoveL 210 to (163.93, -737.64, 0) mm, rotated rx 0 ry 90 rz 0 deg; joints [40.899, -58.772, 133.39, 41.935, -78.434, -10.21]
  MoveL 211 to (163.93, -737.64, 10) mm, rotated rx 0 ry 90 rz 0 deg; joints [40.899, -59.499, 133.41, 42.034, -77.909, -10.694]
  Set speed (1000.0 mm/s)
  MoveL 212 to (145.41, -737.64, 10) mm, rotated rx 0 ry 90 rz 0 deg; joints [41.511, -59.992, 134.485, 42.568, -78.452, -10.419]
  MoveL 213 to (145.41, -737.64, 0) mm, rotated rx 0 ry 90 rz 0 deg; joints [41.511, -59.252, 134.465, 42.471, -78.982, -9.923]
  MoveL 214 to (145.41, -737.64, 0) mm, rotated rx 0 ry 90 rz 0 deg; joints [41.511, -59.252, 134.465, 42.471, -78.982, -9.923]
  Set speed (50.0 mm/s)
  MoveL 215 to (154.89, -701.75, 34.46) mm, rotated rx 0 ry 90 rz 0 deg; joints [39.811, -62.388, 135.736, 41.023, -77.284, -10.841]
  Set speed (1000.0 mm/s)
  MoveL 216 to (154.89, -701.75, 34.46) mm, rotated rx 0 ry 90 rz 0 deg; joints [39.811, -62.388, 135.736, 41.023, -77.284, -10.841]
  MoveL 217 to (154.89, -701.75, 44.46) mm, rotated rx 0 ry 90 rz 0 deg; joints [39.811, -63.127, 135.722, 41.137, -76.716, -11.349]
  Set speed (1000.0 mm/s)
  MoveL 218 to (140.3, -705.32, 44.46) mm, rotated rx 0 ry 90 rz 0 deg; joints [40.436, -63.465, 136.399, 41.714, -77.092, -11.262]
  MoveL 219 to (140.3, -705.32, 34.46) mm, rotated rx 0 ry 90 rz 0 deg; joints [40.436, -62.718, 136.413, 41.6, -77.662, -10.742]
  MoveL 220 to (140.3, -705.32, 34.46) mm, rotated rx 0 ry 90 rz 0 deg; joints [40.436, -62.718, 136.413, 41.6, -77.662, -10.742]
  Set speed (50.0 mm/s)
  MoveL 221 to (126.89, -737.64, 0) mm, rotated rx 0 ry 90 rz 0 deg; joints [42.139, -59.723, 135.525, 43.025, -79.521, -9.634]
  Set speed (1000.0 mm/s)
  MoveL 222 to (126.89, -737.64, 0) mm, rotated rx 0 ry 90 rz 0 deg; joints [42.139, -59.723, 135.525, 43.025, -79.521, -9.634]
  MoveL 223 to (126.89, -737.64, 10) mm, rotated rx 0 ry 90 rz 0 deg; joints [42.139, -60.476, 135.545, 43.12, -78.986, -10.143]
  Set speed (1000.0 mm/s)
  MoveL 224 to (108.36, -737.64, 10) mm, rotated rx 0 ry 90 rz 0 deg; joints [42.783, -60.952, 136.59, 43.691, -79.511, -9.866]
  MoveL 225 to (108.36, -737.64, 0) mm, rotated rx 0 ry 90 rz 0 deg; joints [42.783, -60.185, 136.569, 43.598, -80.051, -9.343]
  MoveL 226 to (108.36, -737.64, 0) mm, rotated rx 0 ry 90 rz 0 deg; joints [42.783, -60.185, 136.569, 43.598, -80.051, -9.343]
  Set speed (50.0 mm/s)
  MoveL 227 to (125.7, -708.89, 34.46) mm, rotated rx 0 ry 90 rz 0 deg; joints [41.07, -63.041, 137.078, 42.189, -78.034, -10.644]
  Set speed (1000.0 mm/s)
  MoveL 228 to (125.7, -708.89, 34.46) mm, rotated rx 0 ry 90 rz 0 deg; joints [41.07, -63.041, 137.078, 42.189, -78.034, -10.644]
  MoveL 229 to (125.7, -708.89, 44.46) mm, rotated rx 0 ry 90 rz 0 deg; joints [41.07, -63.798, 137.063, 42.302, -77.463, -11.174]
  Set speed (1000.0 mm/s)
  MoveL 230 to (111.11, -712.46, 44.46) mm, rotated rx 0 ry 90 rz 0 deg; joints [41.715, -64.124, 137.716, 42.901, -77.828, -11.086]
  MoveL 231 to (111.11, -712.46, 34.46) mm, rotated rx 0 ry 90 rz 0 deg; joints [41.715, -63.358, 137.73, 42.789, -78.399, -10.544]
  MoveL 232 to (111.11, -712.46, 34.46) mm, rotated rx 0 ry 90 rz 0 deg; joints [41.715, -63.358, 137.73, 42.789, -78.399, -10.544]
  Set speed (50.0 mm/s)
  MoveL 233 to (89.84, -737.64, 0) mm, rotated rx 0 ry 90 rz 0 deg; joints [43.442, -60.638, 137.598, 44.19, -80.571, -9.049]
  Set speed (1000.0 mm/s)
  MoveL 234 to (89.84, -737.64, 0) mm, rotated rx 0 ry 90 rz 0 deg; joints [43.442, -60.638, 137.598, 44.19, -80.571, -9.049]
  MoveL 235 to (89.84, -737.64, 10) mm, rotated rx 0 ry 90 rz 0 deg; joints [43.442, -61.418, 137.619, 44.281, -80.027, -9.587]
  Set speed (1000.0 mm/s)
  MoveL 236 to (71.31, -737.64, 10) mm, rotated rx 0 ry 90 rz 0 deg; joints [44.118, -61.876, 138.632, 44.89, -80.533, -9.305]
  MoveL 237 to (71.31, -737.64, 0) mm, rotated rx 0 ry 90 rz 0 deg; joints [44.118, -61.082, 138.611, 44.802, -81.081, -8.753]
  MoveL 238 to (71.31, -737.64, 0) mm, rotated rx 0 ry 90 rz 0 deg; joints [44.118, -61.082, 138.611, 44.802, -81.081, -8.753]
  Set speed (50.0 mm/s)
  MoveL 239 to (96.52, -716.03, 34.46) mm, rotated rx 0 ry 90 rz 0 deg; joints [42.37, -63.669, 138.37, 43.4, -78.759, -10.445]
  Set speed (1000.0 mm/s)
  MoveL 240 to (96.52, -716.03, 34.46) mm, rotated rx 0 ry 90 rz 0 deg; joints [42.37, -63.669, 138.37, 43.4, -78.759, -10.445]
  MoveL 241 to (96.52, -716.03, 44.46) mm, rotated rx 0 ry 90 rz 0 deg; joints [42.37, -64.444, 138.356, 43.511, -78.186, -10.999]
  Set speed (1000.0 mm/s)
  MoveL 242 to (81.92, -719.6, 44.46) mm, rotated rx 0 ry 90 rz 0 deg; joints [43.034, -64.757, 138.983, 44.133, -78.539, -10.911]
  MoveL 243 to (81.92, -719.6, 34.46) mm, rotated rx 0 ry 90 rz 0 deg; joints [43.034, -63.974, 138.998, 44.023, -79.112, -10.346]
  MoveL 244 to (81.92, -719.6, 34.46) mm, rotated rx 0 ry 90 rz 0 deg; joints [43.034, -63.974, 138.998, 44.023, -79.112, -10.346]
  Set speed (50.0 mm/s)
  MoveL 245 to (52.79, -737.64, 0) mm, rotated rx 0 ry 90 rz 0 deg; joints [44.811, -61.516, 139.607, 45.434, -81.582, -8.454]
  Set speed (1000.0 mm/s)
  MoveL 246 to (52.79, -737.64, 0) mm, rotated rx 0 ry 90 rz 0 deg; joints [44.811, -61.516, 139.607, 45.434, -81.582, -8.454]
  MoveL 247 to (52.79, -737.64, 10) mm, rotated rx 0 ry 90 rz 0 deg; joints [44.811, -62.325, 139.629, 45.52, -81.03, -9.022]
  Set speed (1000.0 mm/s)
  MoveL 248 to (34.27, -737.64, 10) mm, rotated rx 0 ry 90 rz 0 deg; joints [45.521, -62.764, 140.61, 46.17, -81.517, -8.736]
  MoveL 249 to (34.27, -737.64, 0) mm, rotated rx 0 ry 90 rz 0 deg; joints [45.521, -61.94, 140.588, 46.087, -82.073, -8.152]
  MoveL 250 to (34.27, -737.64, 0) mm, rotated rx 0 ry 90 rz 0 deg; joints [45.521, -61.94, 140.588, 46.087, -82.073, -8.152]
  Set speed (50.0 mm/s)
  MoveL 251 to (67.33, -723.18, 34.46) mm, rotated rx 0 ry 90 rz 0 deg; joints [43.709, -64.273, 139.613, 44.657, -79.459, -10.246]
  Set speed (1000.0 mm/s)
  MoveL 252 to (67.33, -723.18, 34.46) mm, rotated rx 0 ry 90 rz 0 deg; joints [43.709, -64.273, 139.613, 44.657, -79.459, -10.246]
  MoveL 253 to (67.33, -723.18, 44.46) mm, rotated rx 0 ry 90 rz 0 deg; joints [43.709, -65.065, 139.598, 44.766, -78.886, -10.824]
  Set speed (1000.0 mm/s)
  MoveL 254 to (52.74, -726.75, 44.46) mm, rotated rx 0 ry 90 rz 0 deg; joints [44.395, -65.366, 140.2, 45.41, -79.226, -10.737]
  MoveL 255 to (52.74, -726.75, 34.46) mm, rotated rx 0 ry 90 rz 0 deg; joints [44.395, -64.565, 140.215, 45.303, -79.8, -10.147]
  MoveL 256 to (52.74, -726.75, 34.46) mm, rotated rx 0 ry 90 rz 0 deg; joints [44.395, -64.565, 140.215, 45.303, -79.8, -10.147]
  Set speed (50.0 mm/s)
  MoveL 257 to (15.74, -737.64, 0) mm, rotated rx 0 ry 90 rz 0 deg; joints [46.249, -62.355, 141.553, 46.761, -82.553, -7.848]
  Set speed (1000.0 mm/s)
  MoveL 258 to (15.74, -737.64, 0) mm, rotated rx 0 ry 90 rz 0 deg; joints [46.249, -62.355, 141.553, 46.761, -82.553, -7.848]
  MoveL 259 to (15.74, -737.64, 10) mm, rotated rx 0 ry 90 rz 0 deg; joints [46.249, -63.195, 141.575, 46.841, -81.993, -8.449]
  Set speed (1000.0 mm/s)
  MoveL 260 to (-2.78, -723.28, 10) mm, rotated rx 0 ry 90 rz 0 deg; joints [46.443, -63.959, 143.3, 46.941, -82.678, -7.767]
  MoveL 261 to (-2.78, -723.28, 0) mm, rotated rx 0 ry 90 rz 0 deg; joints [46.443, -63.09, 143.278, 46.865, -83.256, -7.144]
  MoveL 262 to (-2.78, -723.28, 0) mm, rotated rx 0 ry 90 rz 0 deg; joints [46.443, -63.09, 143.278, 46.865, -83.256, -7.144]
  Set speed (50.0 mm/s)
  MoveL 263 to (35.78, -720.65, 34.46) mm, rotated rx 0 ry 90 rz 0 deg; joints [44.808, -65.158, 141.44, 45.637, -80.314, -9.761]
  Set speed (1000.0 mm/s)
  MoveL 264 to (35.78, -720.65, 34.46) mm, rotated rx 0 ry 90 rz 0 deg; joints [44.808, -65.158, 141.44, 45.637, -80.314, -9.761]
  MoveL 265 to (35.78, -720.65, 44.46) mm, rotated rx 0 ry 90 rz 0 deg; joints [44.808, -65.978, 141.425, 45.742, -79.73, -10.368]
  Set speed (1000.0 mm/s)
  MoveL 266 to (33.41, -710.98, 44.46) mm, rotated rx 0 ry 90 rz 0 deg; joints [44.52, -66.295, 142.058, 45.414, -79.901, -10.088]
  MoveL 267 to (33.41, -710.98, 34.46) mm, rotated rx 0 ry 90 rz 0 deg; joints [44.52, -65.465, 142.073, 45.31, -80.495, -9.477]
  MoveL 268 to (33.41, -710.98, 34.46) mm, rotated rx 0 ry 90 rz 0 deg; joints [44.52, -65.465, 142.073, 45.31, -80.495, -9.477]
  Set speed (50.0 mm/s)
  MoveL 269 to (-2.78, -708.91, 0) mm, rotated rx 0 ry 90 rz 0 deg; joints [45.88, -63.415, 144.045, 46.264, -83.492, -6.755]
  Set speed (1000.0 mm/s)
  MoveL 270 to (-2.78, -708.91, 0) mm, rotated rx 0 ry 90 rz 0 deg; joints [45.88, -63.415, 144.045, 46.264, -83.492, -6.755]
  MoveL 271 to (-2.78, -708.91, 10) mm, rotated rx 0 ry 90 rz 0 deg; joints [45.88, -64.296, 144.068, 46.339, -82.899, -7.381]
  Set speed (1000.0 mm/s)
  MoveL 272 to (-2.78, -694.54, 10) mm, rotated rx 0 ry 90 rz 0 deg; joints [45.305, -64.628, 144.826, 45.726, -83.123, -7.002]
  MoveL 273 to (-2.78, -694.54, 0) mm, rotated rx 0 ry 90 rz 0 deg; joints [45.305, -63.733, 144.803, 45.654, -83.732, -6.373]
  MoveL 274 to (-2.78, -694.54, 0) mm, rotated rx 0 ry 90 rz 0 deg; joints [45.305, -63.733, 144.803, 45.654, -83.732, -6.373]
  Set speed (50.0 mm/s)
  MoveL 275 to (31.05, -701.31, 34.46) mm, rotated rx 0 ry 90 rz 0 deg; joints [44.227, -65.769, 142.702, 44.979, -80.676, -9.196]
  Set speed (1000.0 mm/s)
  MoveL 276 to (31.05, -701.31, 34.46) mm, rotated rx 0 ry 90 rz 0 deg; joints [44.227, -65.769, 142.702, 44.979, -80.676, -9.196]
  MoveL 277 to (31.05, -701.31, 44.46) mm, rotated rx 0 ry 90 rz 0 deg; joints [44.227, -66.61, 142.687, 45.082, -80.071, -9.81]
  Set speed (1000.0 mm/s)
  MoveL 278 to (28.68, -691.65, 44.46) mm, rotated rx 0 ry 90 rz 0 deg; joints [43.93, -66.923, 143.312, 44.746, -80.243, -9.535]
  MoveL 279 to (28.68, -691.65, 34.46) mm, rotated rx 0 ry 90 rz 0 deg; joints [43.93, -66.072, 143.328, 44.644, -80.859, -8.917]
  MoveL 280 to (28.68, -691.65, 34.46) mm, rotated rx 0 ry 90 rz 0 deg; joints [43.93, -66.072, 143.328, 44.644, -80.859, -8.917]
  Set speed (50.0 mm/s)
  MoveL 281 to (-2.78, -680.18, 0) mm, rotated rx 0 ry 90 rz 0 deg; joints [44.718, -64.045, 145.551, 45.034, -83.976, -5.998]
  Set speed (1000.0 mm/s)
  MoveL 282 to (-2.78, -680.18, 0) mm, rotated rx 0 ry 90 rz 0 deg; joints [44.718, -64.045, 145.551, 45.034, -83.976, -5.998]
  MoveL 283 to (-2.78, -680.18, 10) mm, rotated rx 0 ry 90 rz 0 deg; joints [44.718, -64.955, 145.575, 45.104, -83.35, -6.63]
  Set speed (1000.0 mm/s)
  MoveL 284 to (-2.78, -665.81, 10) mm, rotated rx 0 ry 90 rz 0 deg; joints [44.119, -65.275, 146.313, 44.471, -83.579, -6.265]
  MoveL 285 to (-2.78, -665.81, 0) mm, rotated rx 0 ry 90 rz 0 deg; joints [44.119, -64.35, 146.289, 44.404, -84.222, -5.631]
  MoveL 286 to (-2.78, -665.81, 0) mm, rotated rx 0 ry 90 rz 0 deg; joints [44.119, -64.35, 146.289, 44.404, -84.222, -5.631]
  Set speed (50.0 mm/s)
  MoveL 287 to (26.31, -681.98, 34.46) mm, rotated rx 0 ry 90 rz 0 deg; joints [43.628, -66.372, 143.95, 44.306, -81.042, -8.641]
  Set speed (1000.0 mm/s)
  MoveL 288 to (26.31, -681.98, 34.46) mm, rotated rx 0 ry 90 rz 0 deg; joints [43.628, -66.372, 143.95, 44.306, -81.042, -8.641]
  MoveL 289 to (26.31, -681.98, 44.46) mm, rotated rx 0 ry 90 rz 0 deg; joints [43.628, -67.234, 143.935, 44.406, -80.415, -9.263]
  Set speed (1000.0 mm/s)
  MoveL 290 to (23.95, -672.31, 44.46) mm, rotated rx 0 ry 90 rz 0 deg; joints [43.32, -67.544, 144.553, 44.062, -80.587, -8.994]
  MoveL 291 to (23.95, -672.31, 34.46) mm, rotated rx 0 ry 90 rz 0 deg; joints [43.32, -66.671, 144.569, 43.964, -81.227, -8.368]
  MoveL 292 to (23.95, -672.31, 34.46) mm, rotated rx 0 ry 90 rz 0 deg; joints [43.32, -66.671, 144.569, 43.964, -81.227, -8.368]
  Set speed (50.0 mm/s)
  MoveL 293 to (-2.78, -651.45, 0) mm, rotated rx 0 ry 90 rz 0 deg; joints [43.508, -64.65, 147.018, 43.763, -84.473, -5.271]
  Set speed (1000.0 mm/s)
  MoveL 294 to (-2.78, -651.45, 0) mm, rotated rx 0 ry 90 rz 0 deg; joints [43.508, -64.65, 147.018, 43.763, -84.473, -5.271]
  MoveL 295 to (-2.78, -651.45, 10) mm, rotated rx 0 ry 90 rz 0 deg; joints [43.508, -65.589, 147.042, 43.828, -83.812, -5.907]
  Set speed (1000.0 mm/s)
  MoveL 296 to (-2.78, -637.08, 10) mm, rotated rx 0 ry 90 rz 0 deg; joints [42.884, -65.898, 147.761, 43.173, -84.047, -5.557]
  MoveL 297 to (-2.78, -637.08, 0) mm, rotated rx 0 ry 90 rz 0 deg; joints [42.884, -64.943, 147.737, 43.111, -84.726, -4.918]
  MoveL 298 to (-2.78, -637.08, 0) mm, rotated rx 0 ry 90 rz 0 deg; joints [42.884, -64.943, 147.737, 43.111, -84.726, -4.918]
  Set speed (50.0 mm/s)
  MoveL 299 to (21.58, -662.64, 34.46) mm, rotated rx 0 ry 90 rz 0 deg; joints [43.008, -66.967, 145.184, 43.617, -81.412, -8.098]
  Set speed (1000.0 mm/s)
  MoveL 300 to (21.58, -662.64, 34.46) mm, rotated rx 0 ry 90 rz 0 deg; joints [43.008, -66.967, 145.184, 43.617, -81.412, -8.098]
  MoveL 301 to (21.58, -662.64, 44.46) mm, rotated rx 0 ry 90 rz 0 deg; joints [43.008, -67.852, 145.168, 43.715, -80.76, -8.728]
  Set speed (1000.0 mm/s)
  MoveL 302 to (19.22, -652.98, 44.46) mm, rotated rx 0 ry 90 rz 0 deg; joints [42.69, -68.158, 145.78, 43.362, -80.934, -8.464]
  MoveL 303 to (19.22, -652.98, 34.46) mm, rotated rx 0 ry 90 rz 0 deg; joints [42.69, -67.262, 145.796, 43.266, -81.598, -7.831]
  MoveL 304 to (19.22, -652.98, 34.46) mm, rotated rx 0 ry 90 rz 0 deg; joints [42.69, -67.262, 145.796, 43.266, -81.598, -7.831]
  Set speed (50.0 mm/s)
  MoveL 305 to (-2.78, -622.72, 0) mm, rotated rx 0 ry 90 rz 0 deg; joints [42.247, -65.23, 148.445, 42.448, -84.983, -4.574]
  Set speed (1000.0 mm/s)
  MoveL 306 to (-2.78, -622.72, 0) mm, rotated rx 0 ry 90 rz 0 deg; joints [42.247, -65.23, 148.445, 42.448, -84.983, -4.574]
  MoveL 307 to (-2.78, -622.72, 10) mm, rotated rx 0 ry 90 rz 0 deg; joints [42.247, -66.2, 148.47, 42.508, -84.285, -5.215]
  Set speed (1000.0 mm/s)
  MoveL 308 to (-2.78, -608.35, 10) mm, rotated rx 0 ry 90 rz 0 deg; joints [41.597, -66.496, 149.168, 41.831, -84.526, -4.88]
  MoveL 309 to (-2.78, -608.35, 0) mm, rotated rx 0 ry 90 rz 0 deg; joints [41.597, -65.511, 149.143, 41.773, -85.242, -4.237]
  MoveL 310 to (-2.78, -608.35, 0) mm, rotated rx 0 ry 90 rz 0 deg; joints [41.597, -65.511, 149.143, 41.773, -85.242, -4.237]
  Set speed (50.0 mm/s)
  MoveL 311 to (16.85, -643.31, 34.46) mm, rotated rx 0 ry 90 rz 0 deg; joints [42.367, -67.555, 146.404, 42.911, -81.785, -7.566]
  Set speed (1000.0 mm/s)
  MoveL 312 to (16.85, -643.31, 34.46) mm, rotated rx 0 ry 90 rz 0 deg; joints [42.367, -67.555, 146.404, 42.911, -81.785, -7.566]
  MoveL 313 to (16.85, -643.31, 44.46) mm, rotated rx 0 ry 90 rz 0 deg; joints [42.367, -68.463, 146.387, 43.006, -81.108, -8.203]
  Set speed (1000.0 mm/s)
  MoveL 314 to (14.49, -633.64, 44.46) mm, rotated rx 0 ry 90 rz 0 deg; joints [42.038, -68.766, 146.992, 42.645, -81.283, -7.946]
  MoveL 315 to (14.49, -633.64, 34.46) mm, rotated rx 0 ry 90 rz 0 deg; joints [42.038, -67.845, 147.008, 42.551, -81.973, -7.305]
  MoveL 316 to (14.49, -633.64, 34.46) mm, rotated rx 0 ry 90 rz 0 deg; joints [42.038, -67.845, 147.008, 42.551, -81.973, -7.305]
  Set speed (50.0 mm/s)
  MoveL 317 to (-2.78, -593.99, 0) mm, rotated rx 0 ry 90 rz 0 deg; joints [40.934, -65.785, 149.831, 41.087, -85.505, -3.909]
  Set speed (1000.0 mm/s)
  MoveL 318 to (-2.78, -593.99, 0) mm, rotated rx 0 ry 90 rz 0 deg; joints [40.934, -65.785, 149.831, 41.087, -85.505, -3.909]
  MoveL 319 to (-2.78, -593.99, 10) mm, rotated rx 0 ry 90 rz 0 deg; joints [40.934, -66.786, 149.856, 41.142, -84.77, -4.553]
  Set speed (1000.0 mm/s)
  MoveL 320 to (-2.78, -579.62, 10) mm, rotated rx 0 ry 90 rz 0 deg; joints [40.257, -67.07, 150.533, 40.441, -85.016, -4.235]
  MoveL 321 to (-2.78, -579.62, 0) mm, rotated rx 0 ry 90 rz 0 deg; joints [40.257, -66.052, 150.507, 40.389, -85.771, -3.59]
  MoveL 322 to (-2.78, -579.62, 0) mm, rotated rx 0 ry 90 rz 0 deg; joints [40.257, -66.052, 150.507, 40.389, -85.771, -3.59]
  Set speed (50.0 mm/s)
  MoveL 323 to (12.12, -623.97, 34.46) mm, rotated rx 0 ry 90 rz 0 deg; joints [41.704, -68.134, 147.609, 42.187, -82.162, -7.046]
  Set speed (1000.0 mm/s)
  MoveL 324 to (12.12, -623.97, 34.46) mm, rotated rx 0 ry 90 rz 0 deg; joints [41.704, -68.134, 147.609, 42.187, -82.162, -7.046]
  MoveL 325 to (12.12, -623.97, 44.46) mm, rotated rx 0 ry 90 rz 0 deg; joints [41.704, -69.067, 147.592, 42.279, -81.459, -7.691]
  Set speed (1000.0 mm/s)
  MoveL 326 to (9.76, -614.31, 44.46) mm, rotated rx 0 ry 90 rz 0 deg; joints [41.364, -69.366, 148.189, 41.908, -81.635, -7.439]
  MoveL 327 to (9.76, -614.31, 34.46) mm, rotated rx 0 ry 90 rz 0 deg; joints [41.364, -68.421, 148.207, 41.818, -82.352, -6.79]
  MoveL 328 to (9.76, -614.31, 34.46) mm, rotated rx 0 ry 90 rz 0 deg; joints [41.364, -68.421, 148.207, 41.818, -82.352, -6.79]
  Set speed (50.0 mm/s)
  MoveL 329 to (-2.78, -565.26, 0) mm, rotated rx 0 ry 90 rz 0 deg; joints [39.566, -66.313, 151.173, 39.679, -86.04, -3.279]
  Set speed (1000.0 mm/s)
  MoveL 330 to (-2.78, -565.26, 0) mm, rotated rx 0 ry 90 rz 0 deg; joints [39.566, -66.313, 151.173, 39.679, -86.04, -3.279]
  MoveL 331 to (-2.78, -565.26, 10) mm, rotated rx 0 ry 90 rz 0 deg; joints [39.566, -67.347, 151.199, 39.728, -85.264, -3.925]
  Set speed (1000.0 mm/s)
  MoveL 332 to (52.74, -726.75, 44.46) mm, rotated rx 0 ry 90 rz 0 deg; joints [44.395, -65.366, 140.2, 45.41, -79.226, -10.737]
  MoveL 333 to (52.74, -726.75, 34.46) mm, rotated rx 0 ry 90 rz 0 deg; joints [44.395, -64.565, 140.215, 45.303, -79.8, -10.147]
  MoveL 334 to (52.74, -726.75, 34.46) mm, rotated rx 0 ry 90 rz 0 deg; joints [44.395, -64.565, 140.215, 45.303, -79.8, -10.147]
  Set speed (50.0 mm/s)
  MoveL 335 to (21.98, -601.07, 34.46) mm, rotated rx 0 ry 90 rz 0 deg; joints [40.279, -68.4, 148.163, 40.733, -82.208, -6.659]
  Set speed (1000.0 mm/s)
  MoveL 336 to (21.98, -601.07, 34.46) mm, rotated rx 0 ry 90 rz 0 deg; joints [40.279, -68.4, 148.163, 40.733, -82.208, -6.659]
  MoveL 337 to (21.98, -601.07, 44.46) mm, rotated rx 0 ry 90 rz 0 deg; joints [40.279, -69.344, 148.146, 40.823, -81.48, -7.294]
  Set speed (1000.0 mm/s)
  MoveL 338 to (67.33, -723.18, 44.46) mm, rotated rx 0 ry 90 rz 0 deg; joints [43.709, -65.065, 139.598, 44.766, -78.886, -10.824]
  MoveL 339 to (67.33, -723.18, 34.46) mm, rotated rx 0 ry 90 rz 0 deg; joints [43.709, -64.273, 139.613, 44.657, -79.459, -10.246]
  MoveL 340 to (67.33, -723.18, 34.46) mm, rotated rx 0 ry 90 rz 0 deg; joints [43.709, -64.273, 139.613, 44.657, -79.459, -10.246]
  Set speed (50.0 mm/s)
  MoveL 341 to (36.58, -597.5, 34.46) mm, rotated rx 0 ry 90 rz 0 deg; joints [39.553, -68.088, 147.513, 40.036, -81.865, -6.78]
  Set speed (1000.0 mm/s)
  MoveL 342 to (36.58, -597.5, 34.46) mm, rotated rx 0 ry 90 rz 0 deg; joints [39.553, -68.088, 147.513, 40.036, -81.865, -6.78]
  MoveL 343 to (36.58, -597.5, 44.46) mm, rotated rx 0 ry 90 rz 0 deg; joints [39.553, -69.018, 147.496, 40.127, -81.14, -7.397]
  Set speed (1000.0 mm/s)
  MoveL 344 to (81.92, -719.6, 44.46) mm, rotated rx 0 ry 90 rz 0 deg; joints [43.034, -64.757, 138.983, 44.133, -78.539, -10.911]
  MoveL 345 to (81.92, -719.6, 34.46) mm, rotated rx 0 ry 90 rz 0 deg; joints [43.034, -63.974, 138.998, 44.023, -79.112, -10.346]
  MoveL 346 to (81.92, -719.6, 34.46) mm, rotated rx 0 ry 90 rz 0 deg; joints [43.034, -63.974, 138.998, 44.023, -79.112, -10.346]
  Set speed (50.0 mm/s)
  MoveL 347 to (51.17, -593.92, 34.46) mm, rotated rx 0 ry 90 rz 0 deg; joints [38.841, -67.769, 146.85, 39.353, -81.516, -6.899]
  Set speed (1000.0 mm/s)
  MoveL 348 to (51.17, -593.92, 34.46) mm, rotated rx 0 ry 90 rz 0 deg; joints [38.841, -67.769, 146.85, 39.353, -81.516, -6.899]
  MoveL 349 to (51.17, -593.92, 44.46) mm, rotated rx 0 ry 90 rz 0 deg; joints [38.841, -68.686, 146.834, 39.445, -80.794, -7.498]
  Set speed (1000.0 mm/s)
  MoveL 350 to (96.52, -716.03, 44.46) mm, rotated rx 0 ry 90 rz 0 deg; joints [42.37, -64.444, 138.356, 43.511, -78.186, -10.999]
  MoveL 351 to (96.52, -716.03, 34.46) mm, rotated rx 0 ry 90 rz 0 deg; joints [42.37, -63.669, 138.37, 43.4, -78.759, -10.445]
  MoveL 352 to (96.52, -716.03, 34.46) mm, rotated rx 0 ry 90 rz 0 deg; joints [42.37, -63.669, 138.37, 43.4, -78.759, -10.445]
  Set speed (50.0 mm/s)
  MoveL 353 to (65.76, -590.35, 34.46) mm, rotated rx 0 ry 90 rz 0 deg; joints [38.142, -67.445, 146.176, 38.685, -81.159, -7.016]
  Set speed (1000.0 mm/s)
  MoveL 354 to (65.76, -590.35, 34.46) mm, rotated rx 0 ry 90 rz 0 deg; joints [38.142, -67.445, 146.176, 38.685, -81.159, -7.016]
  MoveL 355 to (65.76, -590.35, 44.46) mm, rotated rx 0 ry 90 rz 0 deg; joints [38.142, -68.348, 146.159, 38.778, -80.441, -7.599]
  Set speed (1000.0 mm/s)
  MoveL 356 to (111.11, -712.46, 44.46) mm, rotated rx 0 ry 90 rz 0 deg; joints [41.715, -64.124, 137.716, 42.901, -77.828, -11.086]
  MoveL 357 to (111.11, -712.46, 34.46) mm, rotated rx 0 ry 90 rz 0 deg; joints [41.715, -63.358, 137.73, 42.789, -78.399, -10.544]
  MoveL 358 to (111.11, -712.46, 34.46) mm, rotated rx 0 ry 90 rz 0 deg; joints [41.715, -63.358, 137.73, 42.789, -78.399, -10.544]
  Set speed (50.0 mm/s)
  MoveL 359 to (80.36, -586.78, 34.46) mm, rotated rx 0 ry 90 rz 0 deg; joints [37.456, -67.114, 145.489, 38.031, -80.795, -7.132]
  Set speed (1000.0 mm/s)
  MoveL 360 to (80.36, -586.78, 34.46) mm, rotated rx 0 ry 90 rz 0 deg; joints [37.456, -67.114, 145.489, 38.031, -80.795, -7.132]
  MoveL 361 to (80.36, -586.78, 44.46) mm, rotated rx 0 ry 90 rz 0 deg; joints [37.456, -68.004, 145.472, 38.125, -80.082, -7.699]
  Set speed (1000.0 mm/s)
  MoveL 362 to (125.7, -708.89, 44.46) mm, rotated rx 0 ry 90 rz 0 deg; joints [41.07, -63.798, 137.063, 42.302, -77.463, -11.174]
  MoveL 363 to (125.7, -708.89, 34.46) mm, rotated rx 0 ry 90 rz 0 deg; joints [41.07, -63.041, 137.078, 42.189, -78.034, -10.644]
  MoveL 364 to (125.7, -708.89, 34.46) mm, rotated rx 0 ry 90 rz 0 deg; joints [41.07, -63.041, 137.078, 42.189, -78.034, -10.644]
  Set speed (50.0 mm/s)
  MoveL 365 to (94.95, -583.21, 34.46) mm, rotated rx 0 ry 90 rz 0 deg; joints [36.784, -66.777, 144.79, 37.391, -80.425, -7.246]
  Set speed (1000.0 mm/s)
  MoveL 366 to (94.95, -583.21, 34.46) mm, rotated rx 0 ry 90 rz 0 deg; joints [36.784, -66.777, 144.79, 37.391, -80.425, -7.246]
  MoveL 367 to (94.95, -583.21, 44.46) mm, rotated rx 0 ry 90 rz 0 deg; joints [36.784, -67.654, 144.774, 37.486, -79.715, -7.797]
  Set speed (1000.0 mm/s)
  MoveL 368 to (140.3, -705.32, 44.46) mm, rotated rx 0 ry 90 rz 0 deg; joints [40.436, -63.465, 136.399, 41.714, -77.092, -11.262]
  MoveL 369 to (140.3, -705.32, 34.46) mm, rotated rx 0 ry 90 rz 0 deg; joints [40.436, -62.718, 136.413, 41.6, -77.662, -10.742]
  MoveL 370 to (140.3, -705.32, 34.46) mm, rotated rx 0 ry 90 rz 0 deg; joints [40.436, -62.718, 136.413, 41.6, -77.662, -10.742]
  Set speed (50.0 mm/s)
  MoveL 371 to (109.54, -579.64, 34.46) mm, rotated rx 0 ry 90 rz 0 deg; joints [36.124, -66.434, 144.079, 36.765, -80.047, -7.358]
  Set speed (1000.0 mm/s)
  MoveL 372 to (109.54, -579.64, 34.46) mm, rotated rx 0 ry 90 rz 0 deg; joints [36.124, -66.434, 144.079, 36.765, -80.047, -7.358]
  MoveL 373 to (109.54, -579.64, 44.46) mm, rotated rx 0 ry 90 rz 0 deg; joints [36.124, -67.299, 144.063, 36.861, -79.343, -7.894]
  Set speed (1000.0 mm/s)
  MoveL 374 to (154.89, -701.75, 44.46) mm, rotated rx 0 ry 90 rz 0 deg; joints [39.811, -63.127, 135.722, 41.137, -76.716, -11.349]
  MoveL 375 to (154.89, -701.75, 34.46) mm, rotated rx 0 ry 90 rz 0 deg; joints [39.811, -62.388, 135.736, 41.023, -77.284, -10.841]
  MoveL 376 to (154.89, -701.75, 34.46) mm, rotated rx 0 ry 90 rz 0 deg; joints [39.811, -62.388, 135.736, 41.023, -77.284, -10.841]
  Set speed (50.0 mm/s)
  MoveL 377 to (124.14, -576.07, 34.46) mm, rotated rx 0 ry 90 rz 0 deg; joints [35.476, -66.086, 143.357, 36.153, -79.663, -7.469]
  Set speed (1000.0 mm/s)
  MoveL 378 to (124.14, -576.07, 34.46) mm, rotated rx 0 ry 90 rz 0 deg; joints [35.476, -66.086, 143.357, 36.153, -79.663, -7.469]
  MoveL 379 to (124.14, -576.07, 44.46) mm, rotated rx 0 ry 90 rz 0 deg; joints [35.476, -66.937, 143.341, 36.249, -78.964, -7.99]
  Set speed (1000.0 mm/s)
  MoveL 380 to (169.48, -698.18, 44.46) mm, rotated rx 0 ry 90 rz 0 deg; joints [39.197, -62.783, 135.033, 40.572, -76.334, -11.437]
  MoveL 381 to (169.48, -698.18, 34.46) mm, rotated rx 0 ry 90 rz 0 deg; joints [39.197, -62.052, 135.047, 40.457, -76.9, -10.939]
  MoveL 382 to (169.48, -698.18, 34.46) mm, rotated rx 0 ry 90 rz 0 deg; joints [39.197, -62.052, 135.047, 40.457, -76.9, -10.939]
  Set speed (50.0 mm/s)
  MoveL 383 to (138.73, -572.5, 34.46) mm, rotated rx 0 ry 90 rz 0 deg; joints [34.841, -65.731, 142.623, 35.554, -79.273, -7.577]
  Set speed (1000.0 mm/s)
  MoveL 384 to (138.73, -572.5, 34.46) mm, rotated rx 0 ry 90 rz 0 deg; joints [34.841, -65.731, 142.623, 35.554, -79.273, -7.577]
  MoveL 385 to (138.73, -572.5, 44.46) mm, rotated rx 0 ry 90 rz 0 deg; joints [34.841, -66.57, 142.608, 35.651, -78.578, -8.084]
  Set speed (1000.0 mm/s)
  MoveL 386 to (184.08, -694.61, 44.46) mm, rotated rx 0 ry 90 rz 0 deg; joints [38.592, -62.433, 134.332, 40.017, -75.946, -11.524]
  MoveL 387 to (184.08, -694.61, 34.46) mm, rotated rx 0 ry 90 rz 0 deg; joints [38.592, -61.711, 134.346, 39.902, -76.51, -11.037]
  MoveL 388 to (184.08, -694.61, 34.46) mm, rotated rx 0 ry 90 rz 0 deg; joints [38.592, -61.711, 134.346, 39.902, -76.51, -11.037]
  Set speed (50.0 mm/s)
  MoveL 389 to (153.32, -568.93, 34.46) mm, rotated rx 0 ry 90 rz 0 deg; joints [34.218, -65.371, 141.879, 34.968, -78.876, -7.684]
  Set speed (1000.0 mm/s)
  MoveL 390 to (153.32, -568.93, 34.46) mm, rotated rx 0 ry 90 rz 0 deg; joints [34.218, -65.371, 141.879, 34.968, -78.876, -7.684]
  MoveL 391 to (153.32, -568.93, 44.46) mm, rotated rx 0 ry 90 rz 0 deg; joints [34.218, -66.198, 141.863, 35.066, -78.187, -8.177]
  Set speed (1000.0 mm/s)
  MoveL 392 to (198.67, -691.04, 44.46) mm, rotated rx 0 ry 90 rz 0 deg; joints [37.997, -62.077, 133.619, 39.474, -75.552, -11.611]
  MoveL 393 to (198.67, -691.04, 34.46) mm, rotated rx 0 ry 90 rz 0 deg; joints [37.997, -61.363, 133.633, 39.357, -76.114, -11.135]
  MoveL 394 to (198.67, -691.04, 34.46) mm, rotated rx 0 ry 90 rz 0 deg; joints [37.997, -61.363, 133.633, 39.357, -76.114, -11.135]
  Set speed (50.0 mm/s)
  MoveL 395 to (167.92, -565.36, 34.46) mm, rotated rx 0 ry 90 rz 0 deg; joints [33.607, -65.005, 141.123, 34.395, -78.474, -7.789]
  Set speed (1000.0 mm/s)
  MoveL 396 to (167.92, -565.36, 34.46) mm, rotated rx 0 ry 90 rz 0 deg; joints [33.607, -65.005, 141.123, 34.395, -78.474, -7.789]
  MoveL 397 to (167.92, -565.36, 44.46) mm, rotated rx 0 ry 90 rz 0 deg; joints [33.607, -65.82, 141.107, 34.494, -77.789, -8.269]
  Set speed (1000.0 mm/s)
  MoveL 398 to (213.26, -687.47, 44.46) mm, rotated rx 0 ry 90 rz 0 deg; joints [37.412, -61.715, 132.894, 38.941, -75.153, -11.699]
  MoveL 399 to (213.26, -687.47, 34.46) mm, rotated rx 0 ry 90 rz 0 deg; joints [37.412, -61.009, 132.908, 38.824, -75.713, -11.232]
  MoveL 400 to (213.26, -687.47, 34.46) mm, rotated rx 0 ry 90 rz 0 deg; joints [37.412, -61.009, 132.908, 38.824, -75.713, -11.232]
  Set speed (50.0 mm/s)
  MoveL 401 to (182.51, -561.79, 34.46) mm, rotated rx 0 ry 90 rz 0 deg; joints [33.008, -64.633, 140.355, 33.835, -78.065, -7.893]
  Set speed (1000.0 mm/s)
  MoveL 402 to (182.51, -561.79, 34.46) mm, rotated rx 0 ry 90 rz 0 deg; joints [33.008, -64.633, 140.355, 33.835, -78.065, -7.893]
  MoveL 403 to (182.51, -561.79, 44.46) mm, rotated rx 0 ry 90 rz 0 deg; joints [33.008, -65.436, 140.34, 33.934, -77.385, -8.359]
